// TIA Portal V19 export
TYPE "TAx_Speed_STATUSWORD"
// stored: Access Published
   STRUCT
      Enable : Bool;   // 1
      Error : Bool;
      RestartActive : Bool;
      OnlineStartValuesChanged : Bool;   // 0: Restart variable not changed; 1: Restart variable changed, TObject needs to be restarted
      ControlPanelActive : Bool;
      bit_5 : Bool;
      Done : Bool;   // 0: Last Job not done; 1: Last Job Done
      bit_7 : Bool;
      bit_8 : Bool;
      JogCommand : Bool;
      VelocityCommand : Bool;
      bit_11_Reserved : Bool;
      CostantVelocity : Bool;   // 1: Target speed reached;
      Accelerating : Bool;
      Decelerating : Bool;
      bit_15 : Bool;   // 1: Limit switch engaged
      bit_16 : Bool;   // 1: Limit switch engaged
      bit_17 : Bool;   // 1: Limit switch engaged
      bit_18 : Bool;   // 1: Limit switch engaged
      bit_19 : Bool;   // Reserved
      bit_20 : Bool;   // Reserved
      bit_21 : Bool;   // Reserved - 1: Start synchronization with master
      bit_22 : Bool;   // Reserved - 1: Synchronized motion with master
      bit_23 : Bool;
      bit_24 : Bool;
      AxisSimulation : Bool;   // 1: Simulation is active
      TorqueLimitingCommand : Bool;
      InLimitation : Bool;   // 1: Torque limiting is active
      bit_28 : Bool;
      bit_29 : Bool;   // Reserved
      bit_30 : Bool;
      bit_31 : Bool;   // Reserved
   END_STRUCT;
END_TYPE
